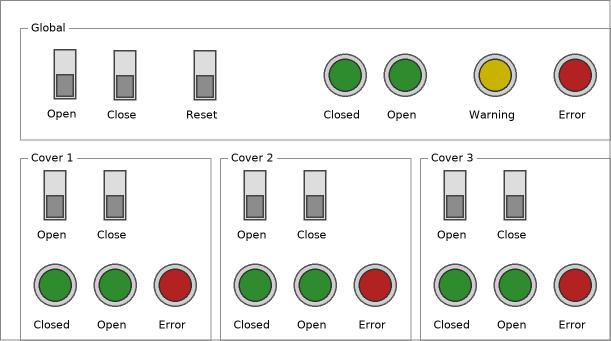
VISUALIZATION Cover  // 611x341
    GroupBox (20,20 591x120), "Global"
        Label (10,79 64x30), "Open"
        DipSwitch (20,29 50x50), variable: MAIN.CoverControl.bOpen, behaviour: TOGGLE, style: Switch-DipSwitch-Gray
        Label (70,80 64x30), "Close"
        DipSwitch (80,30 50x50), variable: MAIN.CoverControl.bClose, behaviour: TOGGLE, style: Switch-DipSwitch-Gray
        Label (150,80 64x30), "Reset"
        DipSwitch (160,30 50x50), variable: MAIN.CoverControl.bReset, behaviour: TOGGLE, style: Switch-DipSwitch-Gray
        Lamp1 (300,30 50x50), variable: MAIN.CoverControl.bAllClosed, style: Lamp-Lamp1-Green
        Label (290,80 64x30), "Closed"
        Lamp1 (360,30 50x50), variable: MAIN.CoverControl.bAllOpen, style: Lamp-Lamp1-Green
        Label (350,80 64x30), "Open"
        Lamp1 (450,30 50x50), variable: MAIN.CoverControl.bWarning, style: Lamp-Lamp1-Yellow
        Label (440,80 64x30), "Warning"
        Lamp1 (530,30 50x50), variable: MAIN.CoverControl.bError, style: Lamp-Lamp1-Red
        Label (520,80 64x30), "Error"
    GroupBox (20,150 191x191), "Cover 1"
        Label (0,70 64x30), "Open"
        Lamp1 (130,110 50x50), variable: MAIN.CoverControl.cover1Error, style: Lamp-Lamp1-Red
        Label (120,160 64x30), "Error"
        DipSwitch (70,20 50x50), variable: MAIN.CoverControl.out_close_cover1, behaviour: TOGGLE, style: Switch-DipSwitch-Gray
        DipSwitch (10,20 50x50), variable: MAIN.CoverControl.out_open_cover1, behaviour: TOGGLE, style: Switch-DipSwitch-Gray
        Label (60,70 64x30), "Close"
        Lamp1 (10,110 50x50), variable: MAIN.CoverControl.cover1Closed, style: Lamp-Lamp1-Green
        Label (0,160 64x30), "Closed"
        Lamp1 (70,110 50x50), variable: MAIN.CoverControl.cover1Open, style: Lamp-Lamp1-Green
        Label (60,160 64x30), "Open"
    GroupBox (220,150 191x191), "Cover 2"
        Label (0,70 64x30), "Open"
        Lamp1 (130,110 50x50), variable: MAIN.CoverControl.cover2Error, style: Lamp-Lamp1-Red
        Label (120,160 64x30), "Error"
        DipSwitch (70,20 50x50), variable: MAIN.CoverControl.outCloseCover2, behaviour: TOGGLE, style: Switch-DipSwitch-Gray
        DipSwitch (10,20 50x50), variable: MAIN.CoverControl.outOpenCover2, behaviour: TOGGLE, style: Switch-DipSwitch-Gray
        Label (60,70 64x30), "Close"
        Lamp1 (10,110 50x50), variable: MAIN.CoverControl.cover2Closed, style: Lamp-Lamp1-Green
        Label (0,160 64x30), "Closed"
        Lamp1 (70,110 50x50), variable: MAIN.CoverControl.cover2Open, style: Lamp-Lamp1-Green
        Label (60,160 64x30), "Open"
    GroupBox (420,150 191x191), "Cover 3"
        Label (0,70 64x30), "Open"
        Lamp1 (130,110 50x50), variable: MAIN.CoverControl.cover3Error, style: Lamp-Lamp1-Red
        Label (120,160 64x30), "Error"
        DipSwitch (70,20 50x50), variable: MAIN.CoverControl.outCloseCover3, behaviour: TOGGLE, style: Switch-DipSwitch-Gray
        DipSwitch (10,20 50x50), variable: MAIN.CoverControl.outOpenCover3, behaviour: TOGGLE, style: Switch-DipSwitch-Gray
        Label (60,70 64x30), "Close"
        Lamp1 (10,110 50x50), variable: MAIN.CoverControl.cover3Closed, style: Lamp-Lamp1-Green
        Label (0,160 64x30), "Closed"
        Lamp1 (70,110 50x50), variable: MAIN.CoverControl.cover3Open, style: Lamp-Lamp1-Green
        Label (60,160 64x30), "Open"
END_VISUALIZATION

(* stored: Version 1.1.0.1, ProductVersion 3.1.4026.8
   Visu Cover: Id {8d36f979-b394-4a24-9a99-523ac5a374ae} *)
